VAR_GLOBAL CONSTANT
	iMaxNumbMovers		: INT := 35;
	iMaxNumbVirtMasters	: INT := 5;
END_VAR

(* stored: Version 1.1.0.1, ProductVersion 3.1.4024.12
   GVL GVL_Constant: Id {0c0a16d8-c818-4096-8edc-bfd15e2b80cc} *)
